ABB RAPID module: Module1.mod

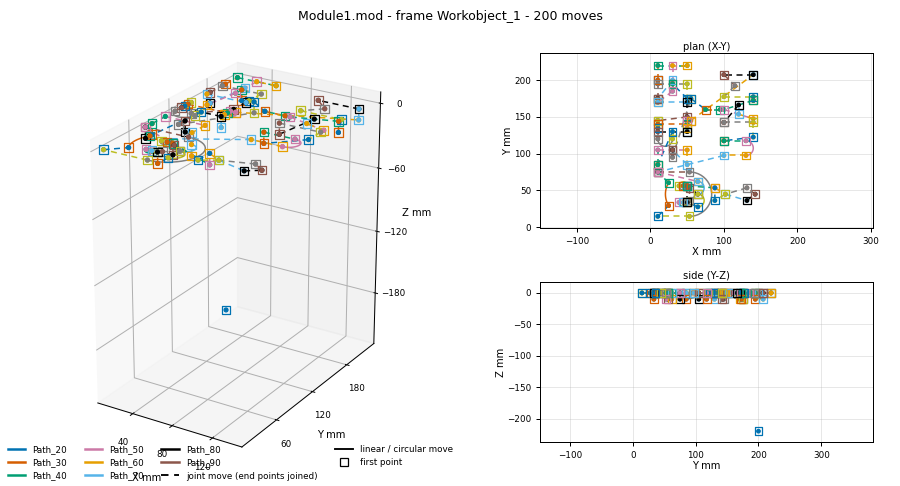
[picture p0: tool path of Module1.mod in frame Workobject_1, 200 of 201 moves have a stored position in this frame; points joined in program order, loops and branches not executed]
MODULE Module1
    CONST robtarget Target_Home:=[[576.159160262,-6.026,569.754077166],[-0.000000007,0,1,0],[0,-1,0,0],[9E+09,9E+09,9E+09,9E+09,9E+09,9E+09]];
    CONST robtarget Target_10:=[[10.001,200,-220],[1,0,0,0],[0,0,0,0],[9E+09,9E+09,9E+09,9E+09,9E+09,9E+09]];
    CONST robtarget Target_20:=[[10.001,200,-0.001],[1,0,0,0],[0,0,0,0],[9E+09,9E+09,9E+09,9E+09,9E+09,9E+09]];
    CONST robtarget Target_30:=[[10.001,220,-0.001],[1,0,0,0],[0,0,0,0],[9E+09,9E+09,9E+09,9E+09,9E+09,9E+09]];
    CONST robtarget Target_40:=[[50.001,220,-0.001],[1,0,0,0],[0,0,0,0],[9E+09,9E+09,9E+09,9E+09,9E+09,9E+09]];
    CONST robtarget Target_50:=[[30.001,220,-0.001],[1,0,0,0],[0,0,0,0],[9E+09,9E+09,9E+09,9E+09,9E+09,9E+09]];
    CONST robtarget Target_60:=[[30.001,200,-0.001],[1,0,0,0],[0,0,0,0],[9E+09,9E+09,9E+09,9E+09,9E+09,9E+09]];
    CONST robtarget Target_70:=[[10.001,175,-10],[1,0,0,0],[0,0,0,0],[9E+09,9E+09,9E+09,9E+09,9E+09,9E+09]];
    CONST robtarget Target_80:=[[10.001,175,-0.001],[1,0,0,0],[0,0,0,0],[9E+09,9E+09,9E+09,9E+09,9E+09,9E+09]];
    CONST robtarget Target_90:=[[10.001,195,-0.001],[1,0,0,0],[0,0,0,0],[9E+09,9E+09,9E+09,9E+09,9E+09,9E+09]];
    CONST robtarget Target_100:=[[50.001,195,-0.001],[1,0,0,0],[0,0,0,0],[9E+09,9E+09,9E+09,9E+09,9E+09,9E+09]];
    CONST robtarget Target_110:=[[50.001,175,-0.001],[1,0,0,0],[0,0,0,0],[9E+09,9E+09,9E+09,9E+09,9E+09,9E+09]];
    CONST robtarget Target_120:=[[29.999,195,-10],[1,0,0,0],[0,0,0,0],[9E+09,9E+09,9E+09,9E+09,9E+09,9E+09]];
    CONST robtarget Target_130:=[[29.999,195,0.001],[1,0,0,0],[0,0,0,0],[9E+09,9E+09,9E+09,9E+09,9E+09,9E+09]];
    CONST robtarget Target_140:=[[29.999,185,0.001],[1,0,0,0],[0,0,0,0],[9E+09,9E+09,9E+09,9E+09,9E+09,9E+09]];
    CONST robtarget Target_150:=[[9.999,170,-10],[1,0,0,0],[0,0,0,0],[9E+09,9E+09,9E+09,9E+09,9E+09,9E+09]];
    CONST robtarget Target_160:=[[9.999,170,0.001],[1,0,0,0],[0,0,0,0],[9E+09,9E+09,9E+09,9E+09,9E+09,9E+09]];
    CONST robtarget Target_170:=[[49.999,170,0.001],[1,0,0,0],[0,0,0,0],[9E+09,9E+09,9E+09,9E+09,9E+09,9E+09]];
    CONST robtarget Target_180:=[[49.999,150,0.001],[1,0,0,0],[0,0,0,0],[9E+09,9E+09,9E+09,9E+09,9E+09,9E+09]];
    CONST robtarget Target_190:=[[9.999,145,-10],[1,0,0,0],[0,0,0,0],[9E+09,9E+09,9E+09,9E+09,9E+09,9E+09]];
    CONST robtarget Target_200:=[[9.999,145,0.001],[1,0,0,0],[0,0,0,0],[9E+09,9E+09,9E+09,9E+09,9E+09,9E+09]];
    CONST robtarget Target_210:=[[9.999,135,0],[1,0,0,0],[0,0,0,0],[9E+09,9E+09,9E+09,9E+09,9E+09,9E+09]];
    CONST robtarget Target_220:=[[9.999,140,0],[1,0,0,0],[0,0,0,0],[9E+09,9E+09,9E+09,9E+09,9E+09,9E+09]];
    CONST robtarget Target_230:=[[49.999,140,0.001],[1,0,0,0],[0,0,0,0],[9E+09,9E+09,9E+09,9E+09,9E+09,9E+09]];
    CONST robtarget Target_240:=[[49.999,145,0.001],[1,0,0,0],[0,0,0,0],[9E+09,9E+09,9E+09,9E+09,9E+09,9E+09]];
    CONST robtarget Target_250:=[[49.999,135,0],[1,0,0,0],[0,0,0,0],[9E+09,9E+09,9E+09,9E+09,9E+09,9E+09]];
    CONST robtarget Target_260:=[[49.999,130,-10],[1,0,0,0],[0,0,0,0],[9E+09,9E+09,9E+09,9E+09,9E+09,9E+09]];
    CONST robtarget Target_270:=[[49.999,130,0],[1,0,0,0],[0,0,0,0],[9E+09,9E+09,9E+09,9E+09,9E+09,9E+09]];
    CONST robtarget Target_280:=[[9.999,130,0],[1,0,0,0],[0,0,0,0],[9E+09,9E+09,9E+09,9E+09,9E+09,9E+09]];
    CONST robtarget Target_290:=[[9.999,120,0],[1,0,0,0],[0,0,0,0],[9E+09,9E+09,9E+09,9E+09,9E+09,9E+09]];
    CONST robtarget Target_300:=[[19.999,110,0],[1,0,0,0],[0,0,0,0],[9E+09,9E+09,9E+09,9E+09,9E+09,9E+09]];
    CONST robtarget Target_310:=[[29.999,120,0],[1,0,0,0],[0,0,0,0],[9E+09,9E+09,9E+09,9E+09,9E+09,9E+09]];
    CONST robtarget Target_320:=[[29.999,130,0],[1,0,0,0],[0,0,0,0],[9E+09,9E+09,9E+09,9E+09,9E+09,9E+09]];
    CONST robtarget Target_330:=[[9.999,85,-10],[1,0,0,0],[0,0,0,0],[9E+09,9E+09,9E+09,9E+09,9E+09,9E+09]];
    CONST robtarget Target_340:=[[9.999,85,0],[1,0,0,0],[0,0,0,0],[9E+09,9E+09,9E+09,9E+09,9E+09,9E+09]];
    CONST robtarget Target_350:=[[9.999,105,0],[1,0,0,0],[0,0,0,0],[9E+09,9E+09,9E+09,9E+09,9E+09,9E+09]];
    CONST robtarget Target_360:=[[49.999,105,0],[1,0,0,0],[0,0,0,0],[9E+09,9E+09,9E+09,9E+09,9E+09,9E+09]];
    CONST robtarget Target_370:=[[49.999,85,0],[1,0,0,0],[0,0,0,0],[9E+09,9E+09,9E+09,9E+09,9E+09,9E+09]];
    CONST robtarget Target_380:=[[29.999,105,-10],[1,0,0,0],[0,0,0,0],[9E+09,9E+09,9E+09,9E+09,9E+09,9E+09]];
    CONST robtarget Target_390:=[[29.999,105,0],[1,0,0,0],[0,0,0,0],[9E+09,9E+09,9E+09,9E+09,9E+09,9E+09]];
    CONST robtarget Target_400:=[[29.999,95,0],[1,0,0,0],[0,0,0,0],[9E+09,9E+09,9E+09,9E+09,9E+09,9E+09]];
    CONST robtarget Target_410:=[[54.999,175,-10],[1,0,0,0],[0,0,0,0],[9E+09,9E+09,9E+09,9E+09,9E+09,9E+09]];
    CONST robtarget Target_420:=[[54.999,175,0.001],[1,0,0,0],[0,0,0,0],[9E+09,9E+09,9E+09,9E+09,9E+09,9E+09]];
    CONST robtarget Target_430:=[[74.999,160,0.001],[1,0,0,0],[0,0,0,0],[9E+09,9E+09,9E+09,9E+09,9E+09,9E+09]];
    CONST robtarget Target_440:=[[94.999,160,0.001],[1,0,0,0],[0,0,0,0],[9E+09,9E+09,9E+09,9E+09,9E+09,9E+09]];
    CONST robtarget Target_450:=[[54.999,145,0.001],[1,0,0,0],[0,0,0,0],[9E+09,9E+09,9E+09,9E+09,9E+09,9E+09]];
    CONST robtarget Target_460:=[[139.999,207.5,-10],[1,0,0,0],[0,0,0,0],[9E+09,9E+09,9E+09,9E+09,9E+09,9E+09]];
    CONST robtarget Target_470:=[[139.999,207.5,0.001],[1,0,0,0],[0,0,0,0],[9E+09,9E+09,9E+09,9E+09,9E+09,9E+09]];
    CONST robtarget Target_480:=[[99.999,207.5,0.001],[1,0,0,0],[0,0,0,0],[9E+09,9E+09,9E+09,9E+09,9E+09,9E+09]];
    CONST robtarget Target_490:=[[114.999,192.5,0.001],[1,0,0,0],[0,0,0,0],[9E+09,9E+09,9E+09,9E+09,9E+09,9E+09]];
    CONST robtarget Target_500:=[[99.999,177.5,0.001],[1,0,0,0],[0,0,0,0],[9E+09,9E+09,9E+09,9E+09,9E+09,9E+09]];
    CONST robtarget Target_510:=[[139.999,177.5,0.001],[1,0,0,0],[0,0,0,0],[9E+09,9E+09,9E+09,9E+09,9E+09,9E+09]];
    CONST robtarget Target_520:=[[139.999,172.5,-10],[1,0,0,0],[0,0,0,0],[9E+09,9E+09,9E+09,9E+09,9E+09,9E+09]];
    CONST robtarget Target_530:=[[139.999,172.5,0.001],[1,0,0,0],[0,0,0,0],[9E+09,9E+09,9E+09,9E+09,9E+09,9E+09]];
    CONST robtarget Target_540:=[[99.999,160,0.001],[1,0,0,0],[0,0,0,0],[9E+09,9E+09,9E+09,9E+09,9E+09,9E+09]];
    CONST robtarget Target_550:=[[139.999,147.5,0.001],[1,0,0,0],[0,0,0,0],[9E+09,9E+09,9E+09,9E+09,9E+09,9E+09]];
    CONST robtarget Target_560:=[[119.999,153.75,0.001],[1,0,0,0],[0,0,0,0],[9E+09,9E+09,9E+09,9E+09,9E+09,9E+09]];
    CONST robtarget Target_570:=[[119.999,166.25,0.001],[1,0,0,0],[0,0,0,0],[9E+09,9E+09,9E+09,9E+09,9E+09,9E+09]];
    CONST robtarget Target_580:=[[99.999,142.5,-10],[1,0,0,0],[0,0,0,0],[9E+09,9E+09,9E+09,9E+09,9E+09,9E+09]];
    CONST robtarget Target_590:=[[99.999,142.5,0.001],[1,0,0,0],[0,0,0,0],[9E+09,9E+09,9E+09,9E+09,9E+09,9E+09]];
    CONST robtarget Target_600:=[[139.999,142.5,0.001],[1,0,0,0],[0,0,0,0],[9E+09,9E+09,9E+09,9E+09,9E+09,9E+09]];
    CONST robtarget Target_610:=[[139.999,122.5,0],[1,0,0,0],[0,0,0,0],[9E+09,9E+09,9E+09,9E+09,9E+09,9E+09]];
    CONST robtarget Target_620:=[[99.999,117.5,-10],[1,0,0,0],[0,0,0,0],[9E+09,9E+09,9E+09,9E+09,9E+09,9E+09]];
    CONST robtarget Target_630:=[[99.999,117.5,0],[1,0,0,0],[0,0,0,0],[9E+09,9E+09,9E+09,9E+09,9E+09,9E+09]];
    CONST robtarget Target_640:=[[129.999,117.5,0],[1,0,0,0],[0,0,0,0],[9E+09,9E+09,9E+09,9E+09,9E+09,9E+09]];
    CONST robtarget Target_650:=[[139.999,107.5,0],[1,0,0,0],[0,0,0,0],[9E+09,9E+09,9E+09,9E+09,9E+09,9E+09]];
    CONST robtarget Target_660:=[[129.999,97.5,0],[1,0,0,0],[0,0,0,0],[9E+09,9E+09,9E+09,9E+09,9E+09,9E+09]];
    CONST robtarget Target_670:=[[99.999,97.5,0],[1,0,0,0],[0,0,0,0],[9E+09,9E+09,9E+09,9E+09,9E+09,9E+09]];
    CONST robtarget Target_680:=[[9.999,75,-10],[1,0,0,0],[0,0,0,0],[9E+09,9E+09,9E+09,9E+09,9E+09,9E+09]];
    CONST robtarget Target_690:=[[9.999,75,0],[1,0,0,0],[0,0,0,0],[9E+09,9E+09,9E+09,9E+09,9E+09,9E+09]];
    CONST robtarget Target_700:=[[53.149,75,0],[1,0,0,0],[0,0,0,0],[9E+09,9E+09,9E+09,9E+09,9E+09,9E+09]];
    CONST robtarget Target_710:=[[83.355,44.795,0],[1,0,0,0],[0,0,0,0],[9E+09,9E+09,9E+09,9E+09,9E+09,9E+09]];
    CONST robtarget Target_720:=[[53.15,14.59,0],[1,0,0,0],[0,0,0,0],[9E+09,9E+09,9E+09,9E+09,9E+09,9E+09]];
    CONST robtarget Target_730:=[[10,14.59,0],[1,0,0,0],[0,0,0,0],[9E+09,9E+09,9E+09,9E+09,9E+09,9E+09]];
    CONST robtarget Target_740:=[[24.645,29.236,0],[1,0,0,0],[0,0,0,0],[9E+09,9E+09,9E+09,9E+09,9E+09,9E+09]];
    CONST robtarget Target_750:=[[20.354,44.795,0],[1,0,0,0],[0,0,0,0],[9E+09,9E+09,9E+09,9E+09,9E+09,9E+09]];
    CONST robtarget Target_760:=[[24.645,60.355,0],[1,0,0,0],[0,0,0,0],[9E+09,9E+09,9E+09,9E+09,9E+09,9E+09]];
    CONST robtarget Target_770:=[[9.999,75,0],[1,0,0,0],[0,0,0,0],[9E+09,9E+09,9E+09,9E+09,9E+09,9E+09]];
    CONST robtarget Target_780:=[[64.466,62.055,-10],[1,0,0,0],[0,0,0,0],[9E+09,9E+09,9E+09,9E+09,9E+09,9E+09]];
    CONST robtarget Target_790:=[[64.466,62.055,0],[1,0,0,0],[0,0,0,0],[9E+09,9E+09,9E+09,9E+09,9E+09,9E+09]];
    CONST robtarget Target_800:=[[73.096,53.425,0],[1,0,0,0],[0,0,0,0],[9E+09,9E+09,9E+09,9E+09,9E+09,9E+09]];
    CONST robtarget Target_810:=[[64.466,44.795,0],[1,0,0,0],[0,0,0,0],[9E+09,9E+09,9E+09,9E+09,9E+09,9E+09]];
    CONST robtarget Target_820:=[[53.149,53.425,0],[1,0,0,0],[0,0,0,0],[9E+09,9E+09,9E+09,9E+09,9E+09,9E+09]];
    CONST robtarget Target_830:=[[53.15,36.165,0],[1,0,0,0],[0,0,0,0],[9E+09,9E+09,9E+09,9E+09,9E+09,9E+09]];
    CONST robtarget Target_840:=[[64.466,44.795,0],[1,0,0,0],[0,0,0,0],[9E+09,9E+09,9E+09,9E+09,9E+09,9E+09]];
    CONST robtarget Target_850:=[[73.096,36.165,0],[1,0,0,0],[0,0,0,0],[9E+09,9E+09,9E+09,9E+09,9E+09,9E+09]];
    CONST robtarget Target_860:=[[64.466,27.535,0],[1,0,0,0],[0,0,0,0],[9E+09,9E+09,9E+09,9E+09,9E+09,9E+09]];
    CONST robtarget Target_870:=[[50.129,33.576,-10],[1,0,0,0],[0,0,0,0],[9E+09,9E+09,9E+09,9E+09,9E+09,9E+09]];
    CONST robtarget Target_880:=[[50.129,33.576,0],[1,0,0,0],[0,0,0,0],[9E+09,9E+09,9E+09,9E+09,9E+09,9E+09]];
    CONST robtarget Target_890:=[[44.544,27.967,0],[1,0,0,0],[0,0,0,0],[9E+09,9E+09,9E+09,9E+09,9E+09,9E+09]];
    CONST robtarget Target_900:=[[38.91,33.576,0],[1,0,0,0],[0,0,0,0],[9E+09,9E+09,9E+09,9E+09,9E+09,9E+09]];
    CONST robtarget Target_910:=[[44.203,39.177,0],[1,0,0,0],[0,0,0,0],[9E+09,9E+09,9E+09,9E+09,9E+09,9E+09]];
    CONST robtarget Target_920:=[[50.129,33.576,0],[1,0,0,0],[0,0,0,0],[9E+09,9E+09,9E+09,9E+09,9E+09,9E+09]];
    CONST robtarget Target_930:=[[47.476,30.776,0],[1,0,0,0],[0,0,0,0],[9E+09,9E+09,9E+09,9E+09,9E+09,9E+09]];
    CONST robtarget Target_940:=[[44.52,33.576,0],[1,0,0,0],[0,0,0,0],[9E+09,9E+09,9E+09,9E+09,9E+09,9E+09]];
    CONST robtarget Target_950:=[[47.207,36.379,0],[1,0,0,0],[0,0,0,0],[9E+09,9E+09,9E+09,9E+09,9E+09,9E+09]];
    CONST robtarget Target_960:=[[50.129,33.543,0],[1,0,0,0],[0,0,0,0],[9E+09,9E+09,9E+09,9E+09,9E+09,9E+09]];
    CONST robtarget Target_970:=[[50.129,56.014,-10],[1,0,0,0],[0,0,0,0],[9E+09,9E+09,9E+09,9E+09,9E+09,9E+09]];
    CONST robtarget Target_980:=[[50.129,56.014,0],[1,0,0,0],[0,0,0,0],[9E+09,9E+09,9E+09,9E+09,9E+09,9E+09]];
    CONST robtarget Target_990:=[[44.473,50.405,0],[1,0,0,0],[0,0,0,0],[9E+09,9E+09,9E+09,9E+09,9E+09,9E+09]];
    CONST robtarget Target_1000:=[[38.91,56.014,0],[1,0,0,0],[0,0,0,0],[9E+09,9E+09,9E+09,9E+09,9E+09,9E+09]];
    CONST robtarget Target_1010:=[[44.395,61.623,0],[1,0,0,0],[0,0,0,0],[9E+09,9E+09,9E+09,9E+09,9E+09,9E+09]];
    CONST robtarget Target_1020:=[[50.129,56.014,0],[1,0,0,0],[0,0,0,0],[9E+09,9E+09,9E+09,9E+09,9E+09,9E+09]];
    CONST robtarget Target_1030:=[[47.188,53.213,0],[1,0,0,0],[0,0,0,0],[9E+09,9E+09,9E+09,9E+09,9E+09,9E+09]];
    CONST robtarget Target_1040:=[[44.519,56.014,0],[1,0,0,0],[0,0,0,0],[9E+09,9E+09,9E+09,9E+09,9E+09,9E+09]];
    CONST robtarget Target_1050:=[[47.478,58.815,0],[1,0,0,0],[0,0,0,0],[9E+09,9E+09,9E+09,9E+09,9E+09,9E+09]];
    CONST robtarget Target_1060:=[[50.129,56.014,0],[1,0,0,0],[0,0,0,0],[9E+09,9E+09,9E+09,9E+09,9E+09,9E+09]];
    CONST robtarget Target_1070:=[[87.669,53.425,-10],[1,0,0,0],[0,0,0,0],[9E+09,9E+09,9E+09,9E+09,9E+09,9E+09]];
    CONST robtarget Target_1080:=[[87.669,53.425,0],[1,0,0,0],[0,0,0,0],[9E+09,9E+09,9E+09,9E+09,9E+09,9E+09]];
    CONST robtarget Target_1090:=[[102.013,44.795,0],[1,0,0,0],[0,0,0,0],[9E+09,9E+09,9E+09,9E+09,9E+09,9E+09]];
    CONST robtarget Target_1100:=[[131.333,36.165,0],[1,0,0,0],[0,0,0,0],[9E+09,9E+09,9E+09,9E+09,9E+09,9E+09]];
    CONST robtarget Target_1110:=[[142.57,44.795,0],[1,0,0,0],[0,0,0,0],[9E+09,9E+09,9E+09,9E+09,9E+09,9E+09]];
    CONST robtarget Target_1120:=[[131.333,53.425,0],[1,0,0,0],[0,0,0,0],[9E+09,9E+09,9E+09,9E+09,9E+09,9E+09]];
    CONST robtarget Target_1130:=[[102.013,44.795,0],[1,0,0,0],[0,0,0,0],[9E+09,9E+09,9E+09,9E+09,9E+09,9E+09]];
    CONST robtarget Target_1140:=[[87.67,36.165,0],[1,0,0,0],[0,0,0,0],[9E+09,9E+09,9E+09,9E+09,9E+09,9E+09]];
    CONST robtarget Target_1150:=[[87.669,53.425,0],[1,0,0,0],[0,0,0,0],[9E+09,9E+09,9E+09,9E+09,9E+09,9E+09]];
!***********************************************************
    !
    ! M?dulo:  Module1
    !
    ! Descripción:
    !   <Introduzca la descripción aquí>
    !
    ! Autor: acer
    !
    ! Versión: 1.0
    !
    !***********************************************************


    !***********************************************************
    !
    ! Procedimiento Main
    !
    !   Este es el punto de entrada de su programa
    !
    !***********************************************************
    PROC main()
        WHILE TRUE DO
            IF DI_01 = 1 THEN
                Set DO_01;
                Path_10;
                Path_20;
                Set DO_02;
                WaitTime 8.0;
                Reset DO_02;
                Path_30;
                Path_40;
                Path_60;
                Path_50;
                Path_70;
                Path_80;
                Path_90;
                Path_100;
                Path_110;
                Path_120;
                Path_130;
                Path_140;
                Path_150;
                Path_160;
                Path_170;
                Path_180;
                Path_190;
                Path_200;
                Path_210;
                Path_220;
                Path_230;
                Path_240;
                Path_250;
                Path_260;
                Path_270;
                Path_280;
                Path_290;
                Path_300;
                Path_310;
                Path_320;
                Path_330;
                Path_340;
                Path_350;
                Path_360;
                Path_370;
                Path_380;
                Path_390;
                Path_400;
                Path_410;
                Path_420;
                Path_430;
                Path_440;
                Path_450;
                Path_460;
                Path_470;
                Path_480;
                Path_490;
                Path_500;
                Path_510;
                Path_520;
                Path_530;
                Path_540;
                Path_550;
                Path_560;
                Path_570;
                Path_580;
                Path_590;
                Path_600;
                Path_610;
                Path_620;
                Path_630;
                Path_640;
                Path_650;
                Path_660;
                Path_670;
                Path_680;
                Path_690;
                Path_700;
                Path_710;
                Path_720;
                Path_730;
                Path_740;
                Path_750;
                Path_760;
                Path_770;
                Path_780;
                Path_790;
                Path_800;
                Path_810;
                Path_820;
                Path_830;
                Path_840;
                Path_850;
                Path_860;
                Path_870;
                Path_880;
                Path_890;
                Path_900;
                Path_910;
                Path_920;
                Path_930;
                Path_940;
                Path_950;
                Path_960;
                Path_970;
                Path_980;
                Path_990;
                Path_1000;
                Path_1010;
                Path_1020;
                Path_20;
                Reset DO_01;
                Set DO_02;
                WaitTime 8.0;
                Reset DO_02;
                Path_10;
            ENDIF
        ENDWHILE
    ENDPROC
    PROC Path_10()
        MoveJ Target_Home,v100,z10,PortaM\WObj:=wobj0;
    ENDPROC
    PROC Path_20()
        MoveJ Target_10,v100,z10,PortaM\WObj:=Workobject_1;
    ENDPROC
    PROC Path_30()
        MoveJ Target_20,v100,z10,PortaM\WObj:=Workobject_1;
        MoveJ Target_30,v100,z10,PortaM\WObj:=Workobject_1;
    ENDPROC
    PROC Path_40()
        MoveJ Target_30,v100,z10,PortaM\WObj:=Workobject_1;
        MoveJ Target_40,v100,z10,PortaM\WObj:=Workobject_1;
    ENDPROC
    PROC Path_50()
        MoveJ Target_50,v100,z10,PortaM\WObj:=Workobject_1;
        MoveJ Target_60,v100,z10,PortaM\WObj:=Workobject_1;
    ENDPROC
    PROC Path_60()
        MoveJ Target_40,v100,z10,PortaM\WObj:=Workobject_1;
        MoveJ Target_50,v100,z10,PortaM\WObj:=Workobject_1;
    ENDPROC
    PROC Path_70()
        MoveJ Target_60,v100,z10,PortaM\WObj:=Workobject_1;
        MoveJ Target_70,v100,z10,PortaM\WObj:=Workobject_1;
    ENDPROC
    PROC Path_80()
        MoveJ Target_70,v100,z10,PortaM\WObj:=Workobject_1;
        MoveJ Target_80,v100,z10,PortaM\WObj:=Workobject_1;
    ENDPROC
    PROC Path_90()
        MoveJ Target_80,v100,z10,PortaM\WObj:=Workobject_1;
        MoveJ Target_90,v100,z10,PortaM\WObj:=Workobject_1;
    ENDPROC
    PROC Path_100()
        MoveJ Target_90,v100,z10,PortaM\WObj:=Workobject_1;
        MoveJ Target_100,v100,z10,PortaM\WObj:=Workobject_1;
    ENDPROC
    PROC Path_110()
        MoveJ Target_100,v100,z10,PortaM\WObj:=Workobject_1;
        MoveJ Target_110,v100,z10,PortaM\WObj:=Workobject_1;
    ENDPROC
    PROC Path_120()
        MoveJ Target_110,v100,z10,PortaM\WObj:=Workobject_1;
        MoveJ Target_120,v100,z10,PortaM\WObj:=Workobject_1;
    ENDPROC
    PROC Path_130()
        MoveJ Target_120,v100,z10,PortaM\WObj:=Workobject_1;
        MoveJ Target_130,v100,z10,PortaM\WObj:=Workobject_1;
    ENDPROC
    PROC Path_140()
        MoveJ Target_130,v100,z10,PortaM\WObj:=Workobject_1;
        MoveJ Target_140,v100,z10,PortaM\WObj:=Workobject_1;
    ENDPROC
    PROC Path_150()
        MoveJ Target_140,v100,z10,PortaM\WObj:=Workobject_1;
        MoveJ Target_150,v100,z10,PortaM\WObj:=Workobject_1;
    ENDPROC
    PROC Path_160()
        MoveJ Target_150,v100,z10,PortaM\WObj:=Workobject_1;
        MoveJ Target_160,v100,z10,PortaM\WObj:=Workobject_1;
    ENDPROC
    PROC Path_170()
        MoveJ Target_160,v100,z10,PortaM\WObj:=Workobject_1;
        MoveJ Target_170,v100,z10,PortaM\WObj:=Workobject_1;
    ENDPROC
    PROC Path_180()
        MoveJ Target_170,v100,z10,PortaM\WObj:=Workobject_1;
        MoveJ Target_180,v100,z10,PortaM\WObj:=Workobject_1;
    ENDPROC
    PROC Path_190()
        MoveJ Target_180,v100,z10,PortaM\WObj:=Workobject_1;
        MoveJ Target_190,v100,z10,PortaM\WObj:=Workobject_1;
    ENDPROC
    PROC Path_200()
        MoveJ Target_190,v100,z10,PortaM\WObj:=Workobject_1;
        MoveJ Target_200,v100,z10,PortaM\WObj:=Workobject_1;
    ENDPROC
    PROC Path_210()
        MoveJ Target_200,v100,z10,PortaM\WObj:=Workobject_1;
        MoveJ Target_210,v100,z10,PortaM\WObj:=Workobject_1;
    ENDPROC
    PROC Path_220()
        MoveJ Target_210,v100,z10,PortaM\WObj:=Workobject_1;
        MoveJ Target_220,v100,z10,PortaM\WObj:=Workobject_1;
    ENDPROC
    PROC Path_230()
        MoveJ Target_220,v100,z10,PortaM\WObj:=Workobject_1;
        MoveJ Target_230,v100,z10,PortaM\WObj:=Workobject_1;
    ENDPROC
    PROC Path_240()
        MoveJ Target_230,v100,z10,PortaM\WObj:=Workobject_1;
        MoveJ Target_240,v100,z10,PortaM\WObj:=Workobject_1;
    ENDPROC
    PROC Path_250()
        MoveJ Target_240,v100,z10,PortaM\WObj:=Workobject_1;
        MoveJ Target_250,v100,z10,PortaM\WObj:=Workobject_1;
    ENDPROC
    PROC Path_260()
        MoveJ Target_250,v100,z10,PortaM\WObj:=Workobject_1;
        MoveJ Target_260,v100,z10,PortaM\WObj:=Workobject_1;
    ENDPROC
    PROC Path_270()
        MoveJ Target_260,v100,z10,PortaM\WObj:=Workobject_1;
        MoveJ Target_270,v100,z10,PortaM\WObj:=Workobject_1;
    ENDPROC
    PROC Path_280()
        MoveJ Target_270,v100,z10,PortaM\WObj:=Workobject_1;
        MoveJ Target_280,v100,z10,PortaM\WObj:=Workobject_1;
    ENDPROC
    PROC Path_290()
        MoveJ Target_280,v100,z10,PortaM\WObj:=Workobject_1;
        MoveJ Target_290,v100,z10,PortaM\WObj:=Workobject_1;
    ENDPROC
    PROC Path_300()
        MoveJ Target_290,v100,z10,PortaM\WObj:=Workobject_1;
        MoveC Target_300, Target_310, v100,z10,PortaM\WObj:=Workobject_1;
    ENDPROC
    PROC Path_310()
        MoveJ Target_310,v100,z10,PortaM\WObj:=Workobject_1;
        MoveJ Target_320,v100,z10,PortaM\WObj:=Workobject_1;
    ENDPROC
    PROC Path_320()
        MoveJ Target_320,v100,z10,PortaM\WObj:=Workobject_1;
        MoveJ Target_330,v100,z10,PortaM\WObj:=Workobject_1;
    ENDPROC
    PROC Path_330()
        MoveJ Target_330,v100,z10,PortaM\WObj:=Workobject_1;
        MoveJ Target_340,v100,z10,PortaM\WObj:=Workobject_1;
    ENDPROC
    PROC Path_340()
        MoveJ Target_340,v100,z10,PortaM\WObj:=Workobject_1;
        MoveJ Target_350,v100,z10,PortaM\WObj:=Workobject_1;
    ENDPROC
    PROC Path_350()
        MoveJ Target_350,v100,z10,PortaM\WObj:=Workobject_1;
        MoveJ Target_360,v100,z10,PortaM\WObj:=Workobject_1;
    ENDPROC
    PROC Path_360()
        MoveJ Target_360,v100,z10,PortaM\WObj:=Workobject_1;
        MoveJ Target_370,v100,z10,PortaM\WObj:=Workobject_1;
    ENDPROC
    PROC Path_370()
        MoveJ Target_370,v100,z10,PortaM\WObj:=Workobject_1;
        MoveJ Target_380,v100,z10,PortaM\WObj:=Workobject_1;
    ENDPROC
    PROC Path_380()
        MoveJ Target_380,v100,z10,PortaM\WObj:=Workobject_1;
        MoveJ Target_390,v100,z10,PortaM\WObj:=Workobject_1;
    ENDPROC
    PROC Path_390()
        MoveJ Target_390,v100,z10,PortaM\WObj:=Workobject_1;
        MoveJ Target_400,v100,z10,PortaM\WObj:=Workobject_1;
    ENDPROC
    PROC Path_400()
        MoveJ Target_400,v100,z10,PortaM\WObj:=Workobject_1;
        MoveJ Target_410,v100,z10,PortaM\WObj:=Workobject_1;
    ENDPROC
    PROC Path_410()
        MoveJ Target_410,v100,z10,PortaM\WObj:=Workobject_1;
        MoveJ Target_420,v100,z10,PortaM\WObj:=Workobject_1;
    ENDPROC
    PROC Path_420()
        MoveJ Target_420,v100,z10,PortaM\WObj:=Workobject_1;
        MoveJ Target_430,v100,z10,PortaM\WObj:=Workobject_1;
    ENDPROC
    PROC Path_430()
        MoveJ Target_430,v100,z10,PortaM\WObj:=Workobject_1;
        MoveJ Target_440,v100,z10,PortaM\WObj:=Workobject_1;
    ENDPROC
    PROC Path_440()
        MoveJ Target_440,v100,z10,PortaM\WObj:=Workobject_1;
        MoveJ Target_430,v100,z10,PortaM\WObj:=Workobject_1;
    ENDPROC
    PROC Path_450()
        MoveJ Target_450,v100,z10,PortaM\WObj:=Workobject_1;
    ENDPROC
    PROC Path_460()
        MoveJ Target_450,v100,z10,PortaM\WObj:=Workobject_1;
        MoveJ Target_460,v100,z10,PortaM\WObj:=Workobject_1;
    ENDPROC
    PROC Path_470()
        MoveJ Target_460,v100,z10,PortaM\WObj:=Workobject_1;
        MoveJ Target_470,v100,z10,PortaM\WObj:=Workobject_1;
    ENDPROC
    PROC Path_480()
        MoveJ Target_470,v100,z10,PortaM\WObj:=Workobject_1;
        MoveJ Target_480,v100,z10,PortaM\WObj:=Workobject_1;
    ENDPROC
    PROC Path_490()
        MoveJ Target_480,v100,z10,PortaM\WObj:=Workobject_1;
        MoveJ Target_490,v100,z10,PortaM\WObj:=Workobject_1;
    ENDPROC
    PROC Path_500()
        MoveJ Target_490,v100,z10,PortaM\WObj:=Workobject_1;
        MoveJ Target_500,v100,z10,PortaM\WObj:=Workobject_1;
    ENDPROC
    PROC Path_510()
        MoveJ Target_500,v100,z10,PortaM\WObj:=Workobject_1;
        MoveJ Target_510,v100,z10,PortaM\WObj:=Workobject_1;
    ENDPROC
    PROC Path_520()
        MoveJ Target_510,v100,z10,PortaM\WObj:=Workobject_1;
        MoveJ Target_520,v100,z10,PortaM\WObj:=Workobject_1;
    ENDPROC
    PROC Path_530()
        MoveJ Target_520,v100,z10,PortaM\WObj:=Workobject_1;
        MoveJ Target_530,v100,z10,PortaM\WObj:=Workobject_1;
    ENDPROC
    PROC Path_540()
        MoveJ Target_530,v100,z10,PortaM\WObj:=Workobject_1;
        MoveJ Target_540,v100,z10,PortaM\WObj:=Workobject_1;
    ENDPROC
    PROC Path_550()
        MoveJ Target_540,v100,z10,PortaM\WObj:=Workobject_1;
        MoveJ Target_550,v100,z10,PortaM\WObj:=Workobject_1;
    ENDPROC
    PROC Path_560()
        MoveJ Target_550,v100,z10,PortaM\WObj:=Workobject_1;
        MoveJ Target_560,v100,z10,PortaM\WObj:=Workobject_1;
    ENDPROC
    PROC Path_570()
        MoveJ Target_560,v100,z10,PortaM\WObj:=Workobject_1;
        MoveJ Target_570,v100,z10,PortaM\WObj:=Workobject_1;
    ENDPROC
    PROC Path_580()
        MoveJ Target_570,v100,z10,PortaM\WObj:=Workobject_1;
        MoveJ Target_580,v100,z10,PortaM\WObj:=Workobject_1;
    ENDPROC
    PROC Path_590()
        MoveJ Target_580,v100,z10,PortaM\WObj:=Workobject_1;
        MoveJ Target_590,v100,z10,PortaM\WObj:=Workobject_1;
    ENDPROC
    PROC Path_600()
        MoveJ Target_590,v100,z10,PortaM\WObj:=Workobject_1;
        MoveJ Target_600,v100,z10,PortaM\WObj:=Workobject_1;
    ENDPROC
    PROC Path_610()
        MoveJ Target_600,v100,z10,PortaM\WObj:=Workobject_1;
        MoveJ Target_610,v100,z10,PortaM\WObj:=Workobject_1;
    ENDPROC
    PROC Path_620()
        MoveJ Target_610,v100,z10,PortaM\WObj:=Workobject_1;
        MoveJ Target_620,v100,z10,PortaM\WObj:=Workobject_1;
    ENDPROC
    PROC Path_630()
        MoveJ Target_620,v100,z10,PortaM\WObj:=Workobject_1;
        MoveJ Target_630,v100,z10,PortaM\WObj:=Workobject_1;
    ENDPROC
    PROC Path_640()
        MoveJ Target_630,v100,z10,PortaM\WObj:=Workobject_1;
        MoveJ Target_640,v100,z10,PortaM\WObj:=Workobject_1;
    ENDPROC
    PROC Path_650()
        MoveJ Target_640,v100,z10,PortaM\WObj:=Workobject_1;
        MoveC Target_650, Target_660, v100,z10,PortaM\WObj:=Workobject_1;
    ENDPROC
    PROC Path_660()
        MoveJ Target_660,v100,z10,PortaM\WObj:=Workobject_1;
        MoveJ Target_670,v100,z10,PortaM\WObj:=Workobject_1;
    ENDPROC
    PROC Path_670()
        MoveJ Target_670,v100,z10,PortaM\WObj:=Workobject_1;
        MoveJ Target_680,v100,z10,PortaM\WObj:=Workobject_1;
    ENDPROC
    PROC Path_680()
        MoveJ Target_680,v100,z10,PortaM\WObj:=Workobject_1;
        MoveJ Target_690,v100,z10,PortaM\WObj:=Workobject_1;
    ENDPROC
    PROC Path_690()
        MoveJ Target_690,v100,z10,PortaM\WObj:=Workobject_1;
        MoveJ Target_700,v100,z10,PortaM\WObj:=Workobject_1;
    ENDPROC
    PROC Path_700()
        MoveJ Target_700,v100,z10,PortaM\WObj:=Workobject_1;
        MoveC Target_710, Target_720, v100,z10,PortaM\WObj:=Workobject_1;
    ENDPROC
    PROC Path_710()
        MoveJ Target_720,v100,z10,PortaM\WObj:=Workobject_1;
        MoveJ Target_730,v100,z10,PortaM\WObj:=Workobject_1;
    ENDPROC
    PROC Path_720()
        MoveJ Target_730,v100,z10,PortaM\WObj:=Workobject_1;
        MoveJ Target_740,v100,z10,PortaM\WObj:=Workobject_1;
    ENDPROC
    PROC Path_730()
        MoveJ Target_740,v100,z10,PortaM\WObj:=Workobject_1;
        MoveC Target_750, Target_760, v100,z10,PortaM\WObj:=Workobject_1;
    ENDPROC
    PROC Path_740()
        MoveJ Target_760,v100,z10,PortaM\WObj:=Workobject_1;
        MoveJ Target_770,v100,z10,PortaM\WObj:=Workobject_1;
    ENDPROC
    PROC Path_750()
        MoveJ Target_770,v100,z10,PortaM\WObj:=Workobject_1;
        MoveJ Target_780,v100,z10,PortaM\WObj:=Workobject_1;
    ENDPROC
    PROC Path_760()
        MoveJ Target_780,v100,z10,PortaM\WObj:=Workobject_1;
        MoveJ Target_790,v100,z10,PortaM\WObj:=Workobject_1;
    ENDPROC
    PROC Path_770()
        MoveJ Target_790,v100,z10,PortaM\WObj:=Workobject_1;
        MoveC Target_800, Target_810, v100,z10,PortaM\WObj:=Workobject_1;
    ENDPROC
    PROC Path_780()
        MoveJ Target_810,v100,z10,PortaM\WObj:=Workobject_1;
        MoveJ Target_820,v100,z10,PortaM\WObj:=Workobject_1;
    ENDPROC
    PROC Path_790()
        MoveJ Target_820,v100,z10,PortaM\WObj:=Workobject_1;
        MoveJ Target_830,v100,z10,PortaM\WObj:=Workobject_1;
    ENDPROC
    PROC Path_800()
        MoveJ Target_830,v100,z10,PortaM\WObj:=Workobject_1;
        MoveJ Target_840,v100,z10,PortaM\WObj:=Workobject_1;
    ENDPROC
    PROC Path_810()
        MoveJ Target_840,v100,z10,PortaM\WObj:=Workobject_1;
        MoveC Target_850, Target_860, v100,z10,PortaM\WObj:=Workobject_1;
    ENDPROC
    PROC Path_820()
        MoveJ Target_860,v100,z10,PortaM\WObj:=Workobject_1;
        MoveJ Target_870,v100,z10,PortaM\WObj:=Workobject_1;
    ENDPROC
    PROC Path_830()
        MoveJ Target_870,v100,z10,PortaM\WObj:=Workobject_1;
        MoveJ Target_880,v100,z10,PortaM\WObj:=Workobject_1;
    ENDPROC
    PROC Path_840()
        MoveJ Target_880,v100,z10,PortaM\WObj:=Workobject_1;
        MoveC Target_890, Target_900, v100,z10,PortaM\WObj:=Workobject_1;
    ENDPROC
    PROC Path_850()
        MoveJ Target_900,v100,z10,PortaM\WObj:=Workobject_1;
        MoveC Target_910, Target_920, v100,z10,PortaM\WObj:=Workobject_1;
    ENDPROC
    PROC Path_860()
        MoveJ Target_920,v100,z10,PortaM\WObj:=Workobject_1;
        MoveC Target_930,Target_940,v100,z10,PortaM\WObj:=Workobject_1;
    ENDPROC
    PROC Path_870()
        MoveJ Target_940,v100,z10,PortaM\WObj:=Workobject_1;
        MoveC Target_950,Target_960,v100,z10,PortaM\WObj:=Workobject_1;
    ENDPROC
    PROC Path_880()
        MoveJ Target_960,v100,z10,PortaM\WObj:=Workobject_1;
        MoveJ Target_970,v100,z10,PortaM\WObj:=Workobject_1;
    ENDPROC
    PROC Path_890()
        MoveJ Target_970,v100,z10,PortaM\WObj:=Workobject_1;
        MoveJ Target_980,v100,z10,PortaM\WObj:=Workobject_1;
    ENDPROC
    PROC Path_900()
        MoveJ Target_980,v100,z10,PortaM\WObj:=Workobject_1;
        MoveC Target_990,Target_1000,v100,z10,PortaM\WObj:=Workobject_1;
    ENDPROC
    PROC Path_910()
        MoveJ Target_1000,v100,z10,PortaM\WObj:=Workobject_1;
        MoveC Target_1010,Target_1020,v100,z10,PortaM\WObj:=Workobject_1;
    ENDPROC
    PROC Path_920()
        MoveJ Target_1020,v100,z10,PortaM\WObj:=Workobject_1;
        MoveC Target_1030,Target_1040,v100,z10,PortaM\WObj:=Workobject_1;
    ENDPROC
    PROC Path_930()
        MoveJ Target_1040,v100,z10,PortaM\WObj:=Workobject_1;
        MoveC Target_1050,Target_1060,v100,z10,PortaM\WObj:=Workobject_1;
    ENDPROC
    PROC Path_940()
        MoveJ Target_1060,v100,z10,PortaM\WObj:=Workobject_1;
        MoveJ Target_1070,v100,z10,PortaM\WObj:=Workobject_1;
    ENDPROC
    PROC Path_950()
        MoveJ Target_1070,v100,z10,PortaM\WObj:=Workobject_1;
        MoveJ Target_1080,v100,z10,PortaM\WObj:=Workobject_1;
    ENDPROC
    PROC Path_960()
        MoveJ Target_1080,v100,z10,PortaM\WObj:=Workobject_1;
        MoveJ Target_1090,v100,z10,PortaM\WObj:=Workobject_1;
    ENDPROC
    PROC Path_970()
        MoveJ Target_1090,v100,z10,PortaM\WObj:=Workobject_1;
        MoveJ Target_1100,v100,z10,PortaM\WObj:=Workobject_1;
    ENDPROC
    PROC Path_980()
        MoveJ Target_1100,v100,z10,PortaM\WObj:=Workobject_1;
        MoveJ Target_1110,v100,z10,PortaM\WObj:=Workobject_1;
    ENDPROC
    PROC Path_990()
        MoveJ Target_1110,v100,z10,PortaM\WObj:=Workobject_1;
        MoveJ Target_1120,v100,z10,PortaM\WObj:=Workobject_1;
    ENDPROC
    PROC Path_1000()
        MoveJ Target_1120,v100,z10,PortaM\WObj:=Workobject_1;
        MoveJ Target_1130,v100,z10,PortaM\WObj:=Workobject_1;
    ENDPROC
    PROC Path_1010()
        MoveJ Target_1130,v100,z10,PortaM\WObj:=Workobject_1;
        MoveJ Target_1140,v100,z10,PortaM\WObj:=Workobject_1;
    ENDPROC
    PROC Path_1020()
        MoveJ Target_1140,v100,z10,PortaM\WObj:=Workobject_1;
        MoveJ Target_1150,v100,z10,PortaM\WObj:=Workobject_1;
    ENDPROC
ENDMODULE
